(* Logix 5000 project; controller cal1615 1756-L62 rev 20.19; software revision 20.05; part 38 of 82 *)
(* tags used below, declared in another part *)
   AFI : BOOL;   // Always False Bit
   FAULT : BOOL;   // Fault AFI
   HMI : BOOL;   // AFI HMI
   metering_roll_alarm : TIMER;
   metering_roll_close : TIMER;
   p01_param_turret_dia_ft : REAL;
   p01r02_do_green_stack_light_lel : BOOL;   // System Outputs Green Stack Light
   p01r02_do_red_stack_light_LINE : BOOL;
   p01r02_do_yellow_stack_light : BOOL;   // System Outputs Yellow Stack Light
   p01r02_timer_half_second_off : TIMER;   // System Misc Control Timer Second Pulse Off
   p01r02_timer_half_second_on : TIMER;   // System Misc Control Timer 1/2 Second Pulse On
   p01r09_pb_global_reset : BOOL;   // System Modes PB: Global Fault Reset
   p01r13_timer_line_start_warning_dwell : TIMER;   // System Line Start Sequence Pre Start Warning Dwell Timer
   p11r30 : routine;   // Zone 1 Temperature Control
   p12r30 : routine;   // Zone 2 Temperature Control
   p20_acc_ctr_prs_input_max : REAL;
   p20_acc_ctr_prs_input_min : REAL;
   p20_acc_ctr_prs_output_max : REAL;
   p20_acc_ctr_prs_output_min : REAL;
   p20_acc_fill_prs_input_max : REAL;
   p20_acc_fill_prs_input_min : REAL;
   p20_acc_fill_prs_output_max : REAL;
   p20_acc_fill_prs_output_min : REAL;
   p20_acc_ten_prs_input_max : REAL;
   p20_acc_ten_prs_input_min : REAL;
   p20_acc_ten_prs_output_max : REAL;
   p20_acc_ten_prs_output_min : REAL;
   p20_ao_acc_ctr_prs : REAL;   // Letoff Analog Output Accumulator Counter Pressure
   p20_ao_acc_fill_prs : REAL;   // Letoff Analog Output Accumulator Fill Pressure
   p20_ao_acc_ten_prs : REAL;   // Letoff Analog Output Accumulator Tension Pressure
   p20_ao_lo_turret_selected_speed : REAL;   // Letoff Letoff Turret VFD Selected Speed
   p20_ao_loa_selected_speed : REAL;   // Letoff Output Selected Speed
   p20_ao_loa_torque : REAL;
   p20_ao_lob_selected_speed : REAL;   // Letoff Letoff B VFD Selected Speed
   p20_ao_lob_torque : REAL;
   p20_di_acc_empty : BOOL;   // Letoff Digital Input Letoff Accumulator Empty Position
   p20_di_acc_full : BOOL;   // Letoff Digital Input Letoff Accumulator Full Control Position
   p20_di_clutch_prs_ok : BOOL;   // Letoff Modes Accumulator Position Mode
   p20_di_lo_turret : acs800_di_normal;   // Letoff Letoff Turret VFD Drive Inputs
   p20_di_loa_active : BOOL;   // Letoff Digital Input Letoff A Active
   p20_dint_to_hmi : DINT[16];   // Letoff Dint to HMI
   p20_do_acc_enable_tension : BOOL;   // Letoff Digital Output Enable Accumulator Lift Tension
   p20_do_acc_high_prs : BOOL;   // Letoff Digital Output Enable Accumulator Lift Pressure
   p20_do_close_nip : BOOL;   // Letoff Digital Output Feedroll Roll Nip Close
   p20_do_enable_lfr_fwd : BOOL;   // Letoff Digital Output Letoff Accumulator Feedroll Forward
   p20_do_enable_lfr_rev : BOOL;   // Letoff Digital Output Letoff Accumulator Feedroll Reverse
   p20_do_engage_lfr_clutch : BOOL;   // Letoff Digital Output Engage Letoff Accumulator Feedroll Clutch
   p20_do_wdr_turret : acs800_do_normal;
   p20_param_lo_turret_gear_ratio : REAL;
   p20_param_loa_gear_ratio : REAL;
   p20_param_lob_gear_ratio : REAL;
   p20_vfd_di_loa : acs800_di_normal;   // Letoff A VFD Inputs
   p20_vfd_di_lob : acs800_di_normal;   // Letoff B VFD Inputs
   p20_vfd_do_loa : acs800_do_normal;   // Letoff A VFD Outputs
   p20_vfd_do_lob : acs800_do_normal;   // Letoff B VFD Outputs
   p20r01 : routine;   // Letoff Main
   p20r02_letoff_dia_ft : REAL;   // Letoff Misc Control Letoff Diameter [ft]
   p20r04 : routine;   // Letoff Ouput
   p20r04_acc_ctr_prs : SYS_SCP;   // Letoff Analog Outputs Accumulator Counter Pressure
   p20r04_acc_fill_prs : SYS_SCP;   // Letoff Analog Output Accumulator Fill Pressure
   p20r04_acc_ten_prs : SYS_SCP;   // Letoff Analog Output Accumulator Tension Pressure
   p20r04_lo_turret_speed_to_vfd : SYS_SPEED_TO_VFD;   // Letoff Outputs Letoff Turret Speed
   p20r04_loa_speed_to_vfd : SYS_SPEED_TO_VFD;   // Letoff Outputs Letoff A Speed
   p20r04_lob_speed_to_vfd : SYS_SPEED_TO_VFD;   // Letoff Outputs Letoff B Speed
   p20r04_timer_fault : TIMER[4];   // Letoff Output Fault Delay
   p20r04_timer_warning : TIMER[4];   // Letoff Output Warning Delay
   p20r05 : routine;   // Letoff Dint to HMI
   p20r05_timer_fault : TIMER[4];   // Letoff Dint to HMI Fault Delay
   p20r05_timer_warning : TIMER[4];   // Letoff Dint to HMI Warning Delay
   p20r09_accumulator_auto : BOOL;   // Letoff Modes Accumulator Auto Mode
   p20r13_status : DINT;   // Letoff Accumulator Fill Status
   p20r15_loa_on : BOOL;   // Letoff Letoff A VFD On
   p20r16_lob_on : BOOL;   // Letoff Letoff B On
   p20r18_index_complete : BOOL;   // Letoff Letoff Turret VFD Index Complete
   retraction_delay_timer : TIMER;
(* P20_Letoff, continued *)

ROUTINE R04_Output   (* ladder *)
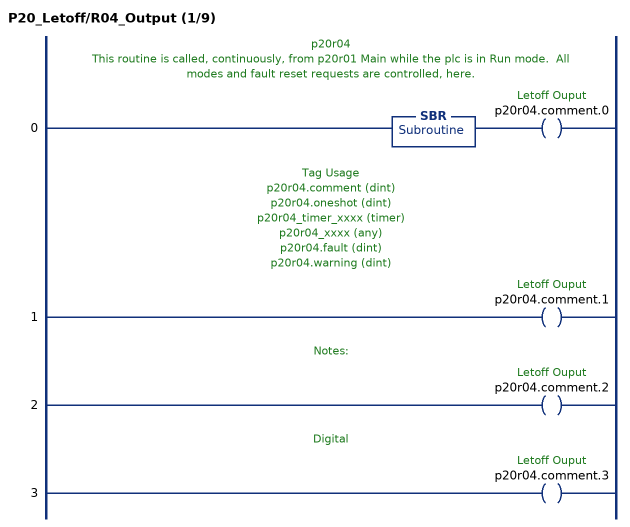
   // p20r04
   // This routine is called, continuously, from p20r01 Main while the plc is in Run mode.  All modes and fault reset requests are controlled, here.
   0: SBR()OTE(p20r04.comment.0);
   // Tag Usage
   // p20r04.comment (dint)
   // p20r04.oneshot (dint)
   // p20r04_timer_xxxx (timer)
   // p20r04_xxxx (any)
   // p20r04.fault (dint)
   // p20r04.warning (dint)
   1: OTE(p20r04.comment.1);
   // Notes:
   2: OTE(p20r04.comment.2);
   // Digital
   3: OTE(p20r04.comment.3);
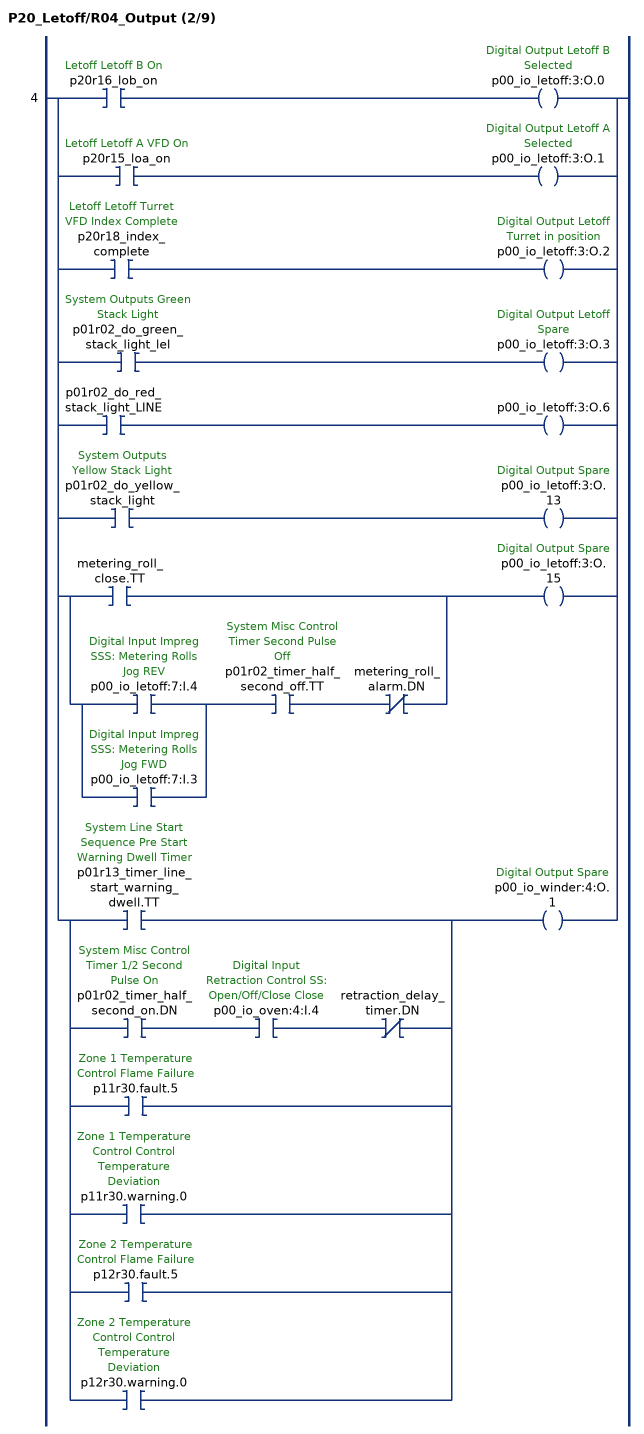
   4: [XIC(p20r16_lob_on) OTE(p00_io_letoff:3:O.0) ,XIC(p20r15_loa_on) OTE(p00_io_letoff:3:O.1) ,XIC(p20r18_index_complete) OTE(p00_io_letoff:3:O.2) ,XIC(p01r02_do_green_stack_light_lel) OTE(p00_io_letoff:3:O.3) ,XIC(p01r02_do_red_stack_light_LINE) OTE(p00_io_letoff:3:O.6) ,[XIC(p01r02_do_yellow_stack_light) OTE(p00_io_letoff:3:O.13) ,[[XIC(metering_roll_close.TT) ,[XIC(p00_io_letoff:7:I.4) ,XIC(p00_io_letoff:7:I.3) ] XIC(p01r02_timer_half_second_off.TT) XIO(metering_roll_alarm.DN) ] OTE(p00_io_letoff:3:O.15) ,[XIC(p01r13_timer_line_start_warning_dwell.TT) ,XIC(p01r02_timer_half_second_on.DN) XIC(p00_io_oven:4:I.4) XIO(retraction_delay_timer.DN) ,XIC(p11r30.fault.5) ,XIC(p11r30.warning.0) ,XIC(p12r30.fault.5) ,XIC(p12r30.warning.0) ] OTE(p00_io_winder:4:O.1) ] ] ];
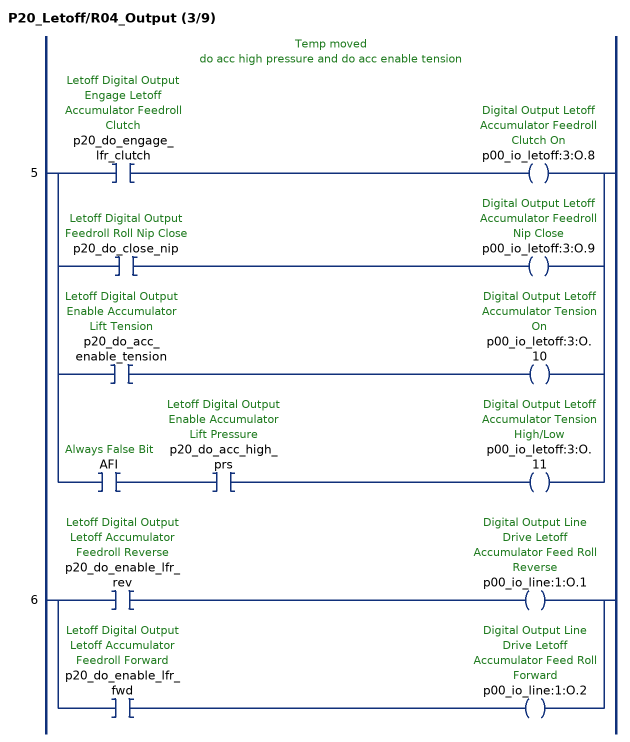
   // Temp moved
   // do acc high pressure and do acc enable tension
   5: [XIC(p20_do_engage_lfr_clutch) OTE(p00_io_letoff:3:O.8) ,XIC(p20_do_close_nip) OTE(p00_io_letoff:3:O.9) ,XIC(p20_do_acc_enable_tension) OTE(p00_io_letoff:3:O.10) ,XIC(AFI) XIC(p20_do_acc_high_prs) OTE(p00_io_letoff:3:O.11) ];
   6: [XIC(p20_do_enable_lfr_rev) OTE(p00_io_line:1:O.1) ,XIC(p20_do_enable_lfr_fwd) OTE(p00_io_line:1:O.2) ];
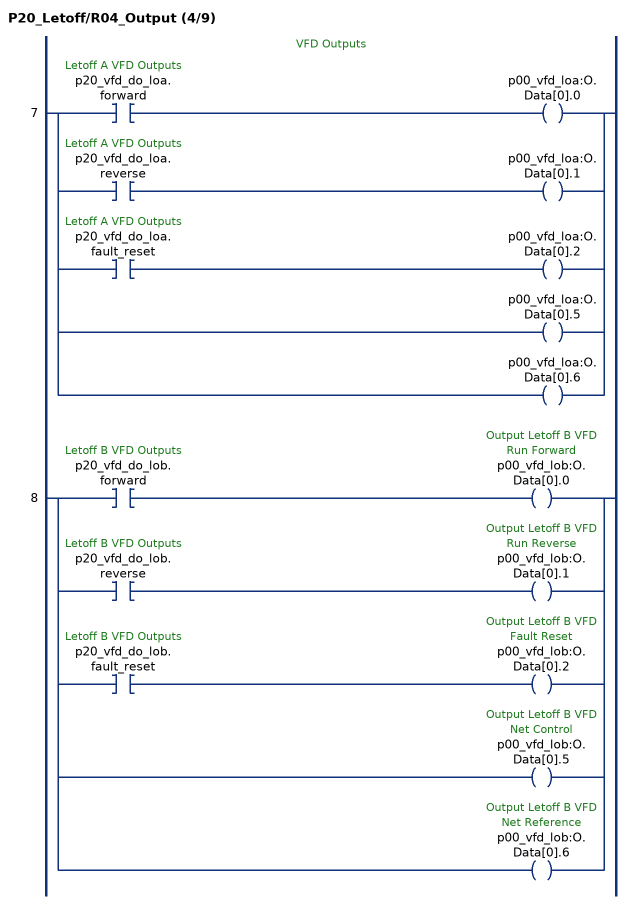
   // VFD Outputs
   7: [XIC(p20_vfd_do_loa.forward) OTE(p00_vfd_loa:O.Data[0].0) ,XIC(p20_vfd_do_loa.reverse) OTE(p00_vfd_loa:O.Data[0].1) ,XIC(p20_vfd_do_loa.fault_reset) OTE(p00_vfd_loa:O.Data[0].2) ,OTE(p00_vfd_loa:O.Data[0].5) ,OTE(p00_vfd_loa:O.Data[0].6) ];
   8: [XIC(p20_vfd_do_lob.forward) OTE(p00_vfd_lob:O.Data[0].0) ,XIC(p20_vfd_do_lob.reverse) OTE(p00_vfd_lob:O.Data[0].1) ,XIC(p20_vfd_do_lob.fault_reset) OTE(p00_vfd_lob:O.Data[0].2) ,OTE(p00_vfd_lob:O.Data[0].5) ,OTE(p00_vfd_lob:O.Data[0].6) ];
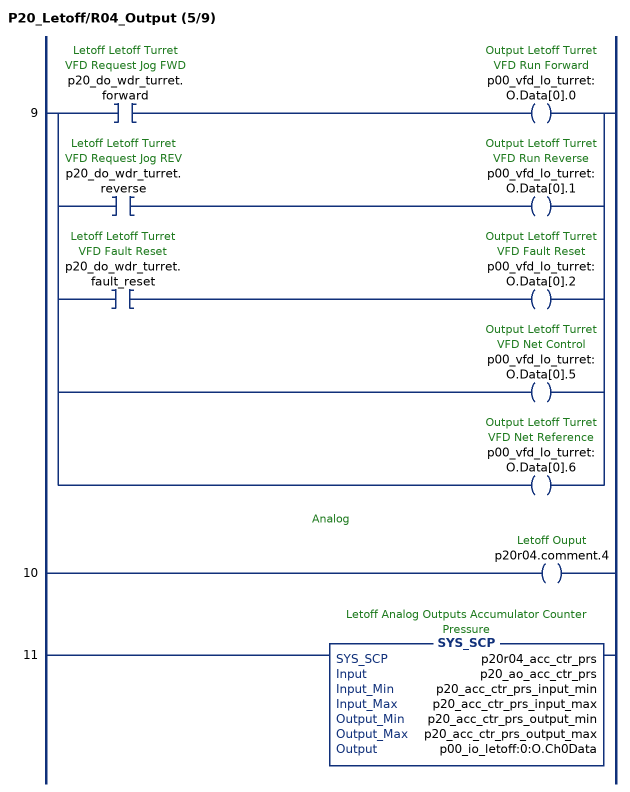
   9: [XIC(p20_do_wdr_turret.forward) OTE(p00_vfd_lo_turret:O.Data[0].0) ,XIC(p20_do_wdr_turret.reverse) OTE(p00_vfd_lo_turret:O.Data[0].1) ,XIC(p20_do_wdr_turret.fault_reset) OTE(p00_vfd_lo_turret:O.Data[0].2) ,OTE(p00_vfd_lo_turret:O.Data[0].5) ,OTE(p00_vfd_lo_turret:O.Data[0].6) ];
   // Analog
   10: OTE(p20r04.comment.4);
   11: SYS_SCP(p20r04_acc_ctr_prs,p20_ao_acc_ctr_prs,p20_acc_ctr_prs_input_min,p20_acc_ctr_prs_input_max,p20_acc_ctr_prs_output_min,p20_acc_ctr_prs_output_max,p00_io_letoff:0:O.Ch0Data);
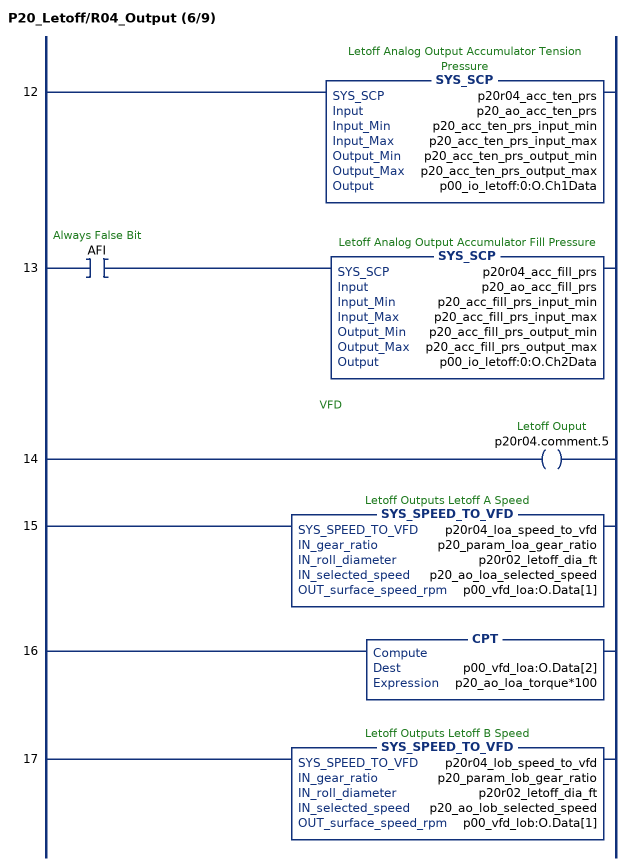
   12: SYS_SCP(p20r04_acc_ten_prs,p20_ao_acc_ten_prs,p20_acc_ten_prs_input_min,p20_acc_ten_prs_input_max,p20_acc_ten_prs_output_min,p20_acc_ten_prs_output_max,p00_io_letoff:0:O.Ch1Data);
   13: XIC(AFI)SYS_SCP(p20r04_acc_fill_prs,p20_ao_acc_fill_prs,p20_acc_fill_prs_input_min,p20_acc_fill_prs_input_max,p20_acc_fill_prs_output_min,p20_acc_fill_prs_output_max,p00_io_letoff:0:O.Ch2Data);
   // VFD
   14: OTE(p20r04.comment.5);
   15: SYS_SPEED_TO_VFD(p20r04_loa_speed_to_vfd,p20_param_loa_gear_ratio,p20r02_letoff_dia_ft,p20_ao_loa_selected_speed,p00_vfd_loa:O.Data[1]);
   16: CPT(p00_vfd_loa:O.Data[2],p20_ao_loa_torque*100);
   17: SYS_SPEED_TO_VFD(p20r04_lob_speed_to_vfd,p20_param_lob_gear_ratio,p20r02_letoff_dia_ft,p20_ao_lob_selected_speed,p00_vfd_lob:O.Data[1]);
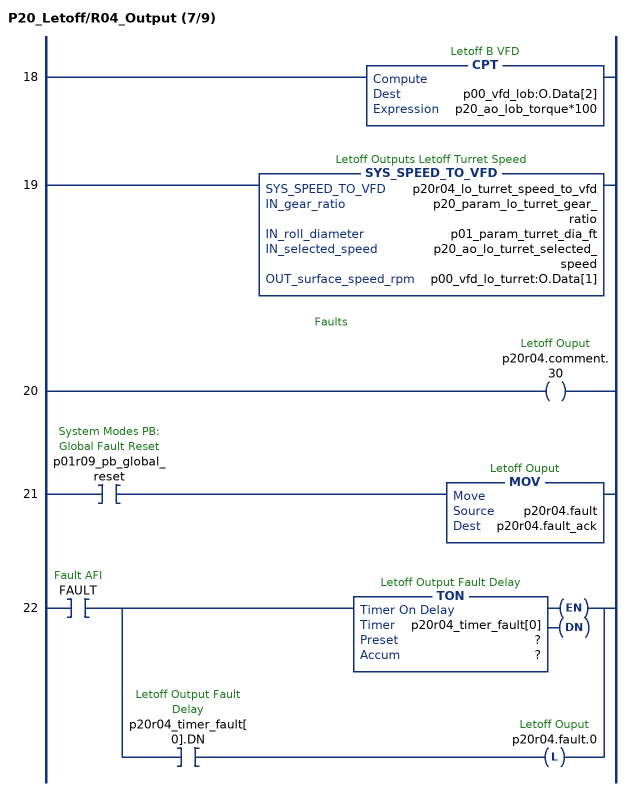
   18: CPT(p00_vfd_lob:O.Data[2],p20_ao_lob_torque*100);
   19: SYS_SPEED_TO_VFD(p20r04_lo_turret_speed_to_vfd,p20_param_lo_turret_gear_ratio,p01_param_turret_dia_ft,p20_ao_lo_turret_selected_speed,p00_vfd_lo_turret:O.Data[1]);
   // Faults
   20: OTE(p20r04.comment.30);
   21: XIC(p01r09_pb_global_reset)MOV(p20r04.fault,p20r04.fault_ack);
   22: XIC(FAULT)[TON(p20r04_timer_fault[0],?,?) ,XIC(p20r04_timer_fault[0].DN) OTL(p20r04.fault.0) ];
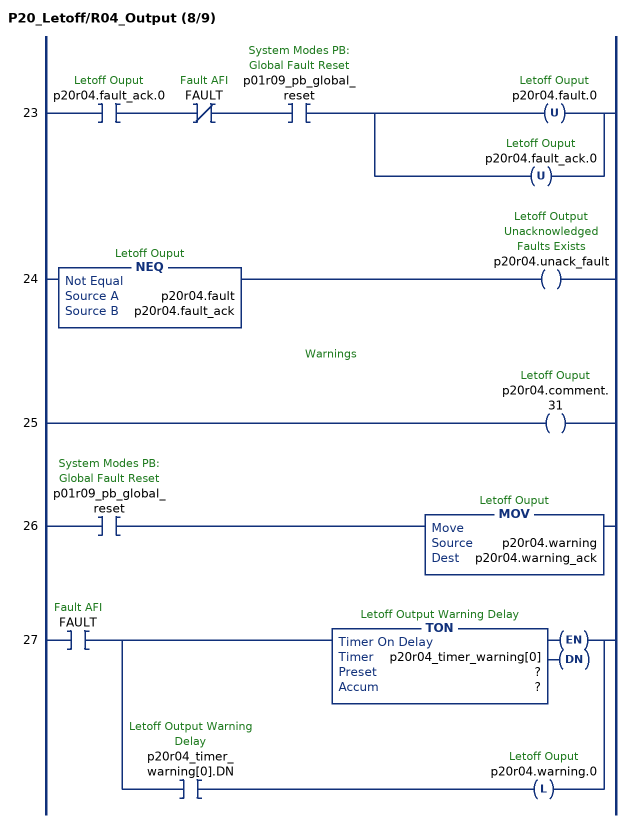
   23: XIC(p20r04.fault_ack.0)XIO(FAULT)XIC(p01r09_pb_global_reset)[OTU(p20r04.fault.0) ,OTU(p20r04.fault_ack.0) ];
   24: NEQ(p20r04.fault,p20r04.fault_ack)OTE(p20r04.unack_fault);
   // Warnings
   25: OTE(p20r04.comment.31);
   26: XIC(p01r09_pb_global_reset)MOV(p20r04.warning,p20r04.warning_ack);
   27: XIC(FAULT)[TON(p20r04_timer_warning[0],?,?) ,XIC(p20r04_timer_warning[0].DN) OTL(p20r04.warning.0) ];
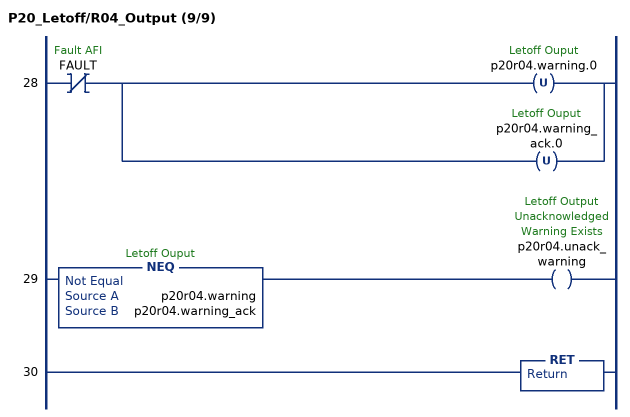
   28: XIO(FAULT)[OTU(p20r04.warning.0) ,OTU(p20r04.warning_ack.0) ];
   29: NEQ(p20r04.warning,p20r04.warning_ack)OTE(p20r04.unack_warning);
   30: RET();
END_ROUTINE

ROUTINE R05_Dint_to_HMI   (* ladder *)
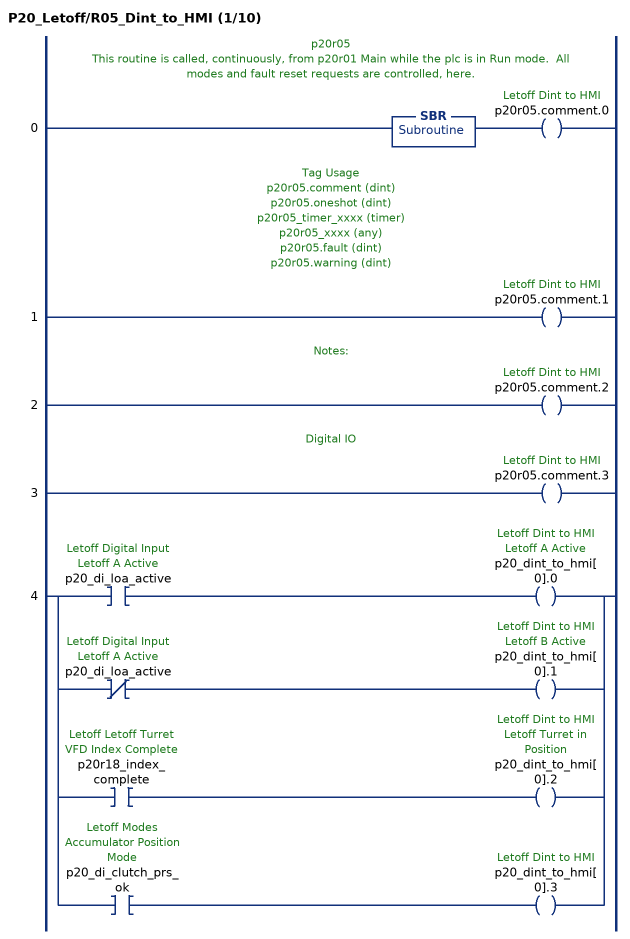
   // p20r05
   // This routine is called, continuously, from p20r01 Main while the plc is in Run mode.  All modes and fault reset requests are controlled, here.
   0: SBR()OTE(p20r05.comment.0);
   // Tag Usage
   // p20r05.comment (dint)
   // p20r05.oneshot (dint)
   // p20r05_timer_xxxx (timer)
   // p20r05_xxxx (any)
   // p20r05.fault (dint)
   // p20r05.warning (dint)
   1: OTE(p20r05.comment.1);
   // Notes:
   2: OTE(p20r05.comment.2);
   // Digital IO
   3: OTE(p20r05.comment.3);
   4: [XIC(p20_di_loa_active) OTE(p20_dint_to_hmi[0].0) ,XIO(p20_di_loa_active) OTE(p20_dint_to_hmi[0].1) ,XIC(p20r18_index_complete) OTE(p20_dint_to_hmi[0].2) ,XIC(p20_di_clutch_prs_ok) OTE(p20_dint_to_hmi[0].3) ];
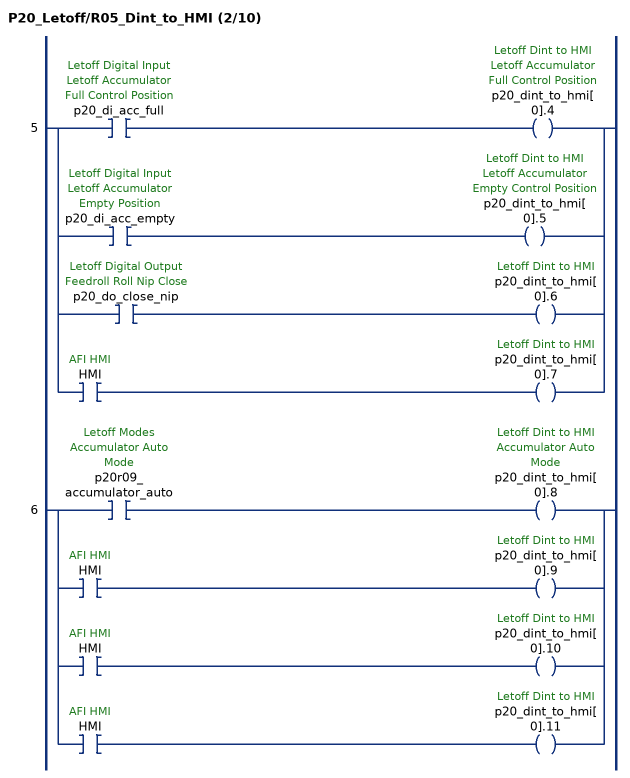
   5: [XIC(p20_di_acc_full) OTE(p20_dint_to_hmi[0].4) ,XIC(p20_di_acc_empty) OTE(p20_dint_to_hmi[0].5) ,XIC(p20_do_close_nip) OTE(p20_dint_to_hmi[0].6) ,XIC(HMI) OTE(p20_dint_to_hmi[0].7) ];
   6: [XIC(p20r09_accumulator_auto) OTE(p20_dint_to_hmi[0].8) ,XIC(HMI) OTE(p20_dint_to_hmi[0].9) ,XIC(HMI) OTE(p20_dint_to_hmi[0].10) ,XIC(HMI) OTE(p20_dint_to_hmi[0].11) ];
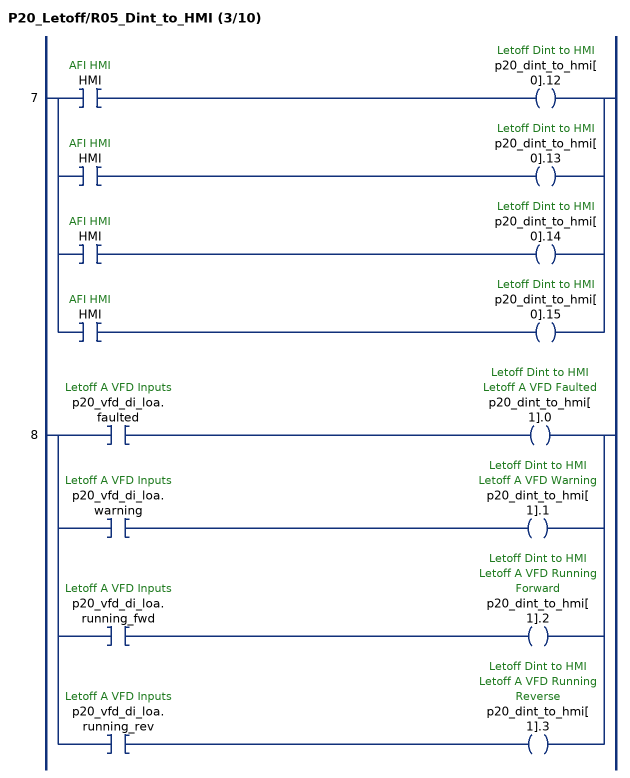
   7: [XIC(HMI) OTE(p20_dint_to_hmi[0].12) ,XIC(HMI) OTE(p20_dint_to_hmi[0].13) ,XIC(HMI) OTE(p20_dint_to_hmi[0].14) ,XIC(HMI) OTE(p20_dint_to_hmi[0].15) ];
   8: [XIC(p20_vfd_di_loa.faulted) OTE(p20_dint_to_hmi[1].0) ,XIC(p20_vfd_di_loa.warning) OTE(p20_dint_to_hmi[1].1) ,XIC(p20_vfd_di_loa.running_fwd) OTE(p20_dint_to_hmi[1].2) ,XIC(p20_vfd_di_loa.running_rev) OTE(p20_dint_to_hmi[1].3) ];
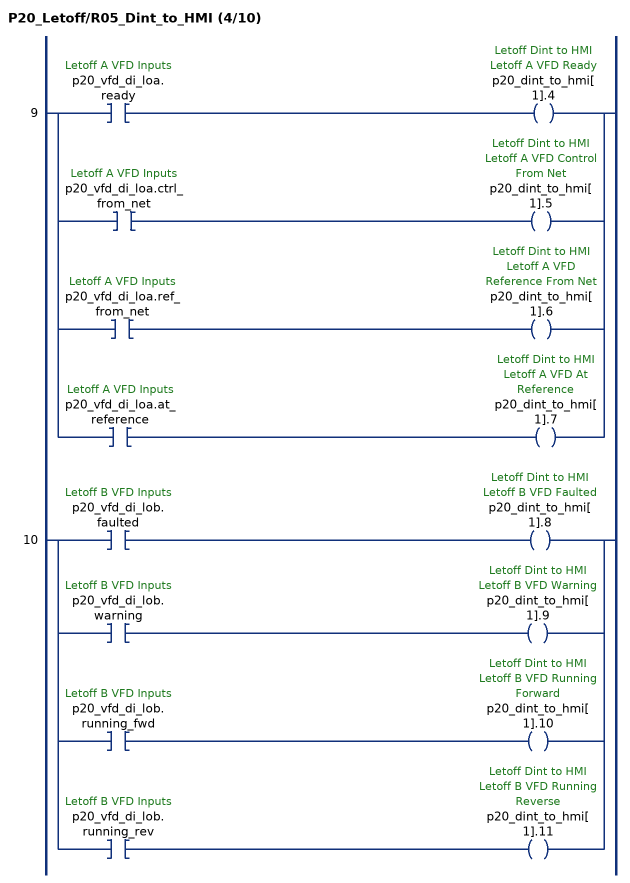
   9: [XIC(p20_vfd_di_loa.ready) OTE(p20_dint_to_hmi[1].4) ,XIC(p20_vfd_di_loa.ctrl_from_net) OTE(p20_dint_to_hmi[1].5) ,XIC(p20_vfd_di_loa.ref_from_net) OTE(p20_dint_to_hmi[1].6) ,XIC(p20_vfd_di_loa.at_reference) OTE(p20_dint_to_hmi[1].7) ];
   10: [XIC(p20_vfd_di_lob.faulted) OTE(p20_dint_to_hmi[1].8) ,XIC(p20_vfd_di_lob.warning) OTE(p20_dint_to_hmi[1].9) ,XIC(p20_vfd_di_lob.running_fwd) OTE(p20_dint_to_hmi[1].10) ,XIC(p20_vfd_di_lob.running_rev) OTE(p20_dint_to_hmi[1].11) ];
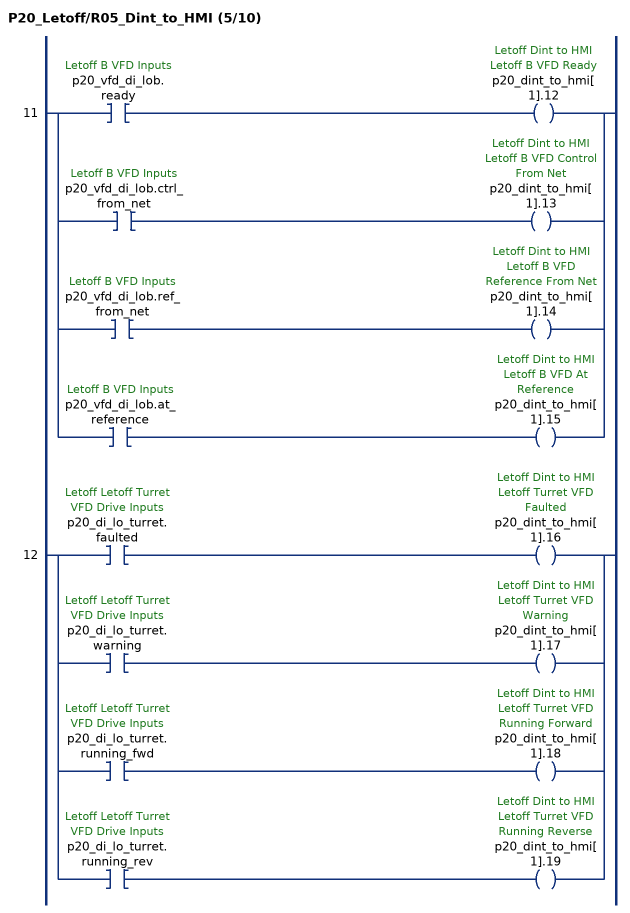
   11: [XIC(p20_vfd_di_lob.ready) OTE(p20_dint_to_hmi[1].12) ,XIC(p20_vfd_di_lob.ctrl_from_net) OTE(p20_dint_to_hmi[1].13) ,XIC(p20_vfd_di_lob.ref_from_net) OTE(p20_dint_to_hmi[1].14) ,XIC(p20_vfd_di_lob.at_reference) OTE(p20_dint_to_hmi[1].15) ];
   12: [XIC(p20_di_lo_turret.faulted) OTE(p20_dint_to_hmi[1].16) ,XIC(p20_di_lo_turret.warning) OTE(p20_dint_to_hmi[1].17) ,XIC(p20_di_lo_turret.running_fwd) OTE(p20_dint_to_hmi[1].18) ,XIC(p20_di_lo_turret.running_rev) OTE(p20_dint_to_hmi[1].19) ];
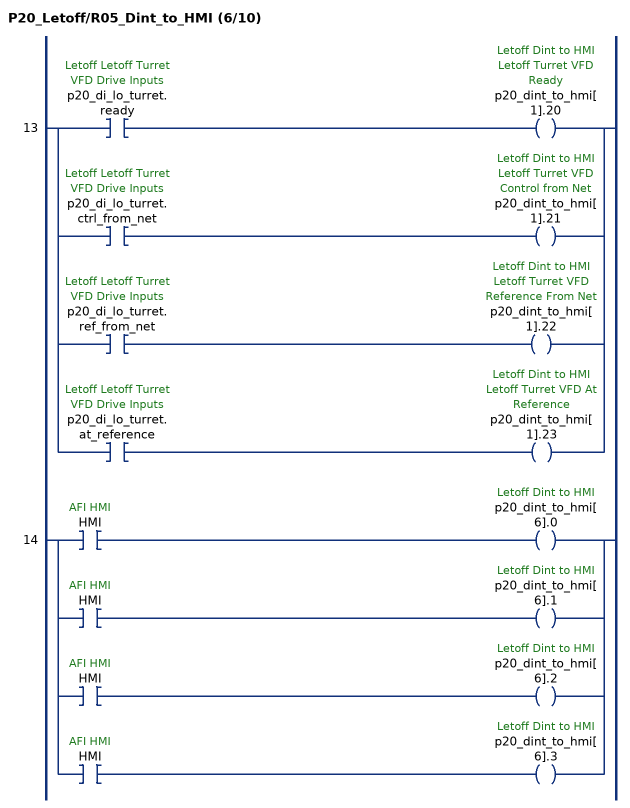
   13: [XIC(p20_di_lo_turret.ready) OTE(p20_dint_to_hmi[1].20) ,XIC(p20_di_lo_turret.ctrl_from_net) OTE(p20_dint_to_hmi[1].21) ,XIC(p20_di_lo_turret.ref_from_net) OTE(p20_dint_to_hmi[1].22) ,XIC(p20_di_lo_turret.at_reference) OTE(p20_dint_to_hmi[1].23) ];
   14: [XIC(HMI) OTE(p20_dint_to_hmi[6].0) ,XIC(HMI) OTE(p20_dint_to_hmi[6].1) ,XIC(HMI) OTE(p20_dint_to_hmi[6].2) ,XIC(HMI) OTE(p20_dint_to_hmi[6].3) ];
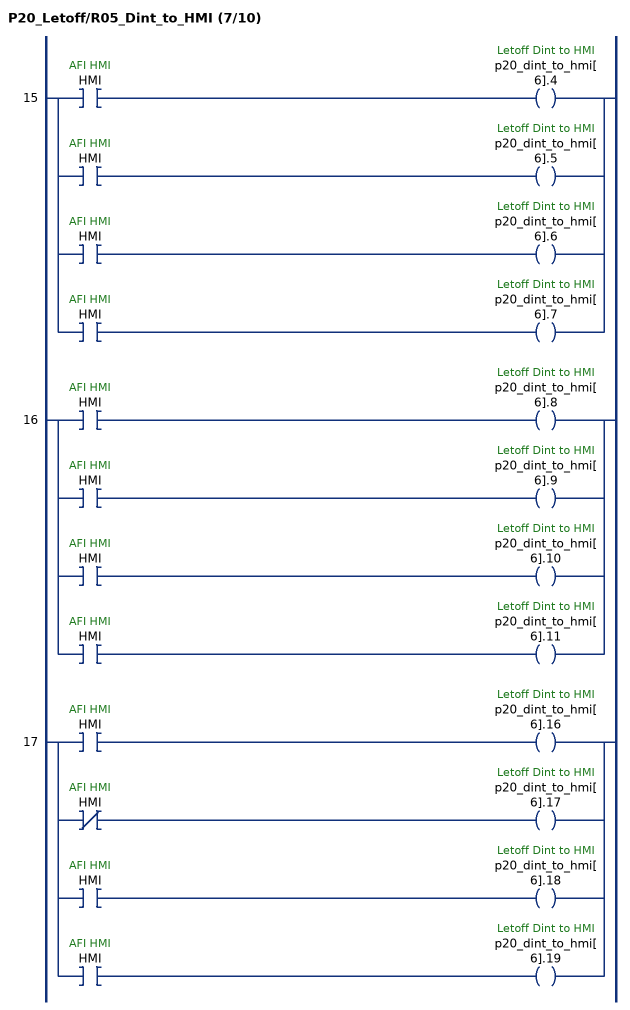
   15: [XIC(HMI) OTE(p20_dint_to_hmi[6].4) ,XIC(HMI) OTE(p20_dint_to_hmi[6].5) ,XIC(HMI) OTE(p20_dint_to_hmi[6].6) ,XIC(HMI) OTE(p20_dint_to_hmi[6].7) ];
   16: [XIC(HMI) OTE(p20_dint_to_hmi[6].8) ,XIC(HMI) OTE(p20_dint_to_hmi[6].9) ,XIC(HMI) OTE(p20_dint_to_hmi[6].10) ,XIC(HMI) OTE(p20_dint_to_hmi[6].11) ];
   17: [XIC(HMI) OTE(p20_dint_to_hmi[6].16) ,XIO(HMI) OTE(p20_dint_to_hmi[6].17) ,XIC(HMI) OTE(p20_dint_to_hmi[6].18) ,XIC(HMI) OTE(p20_dint_to_hmi[6].19) ];
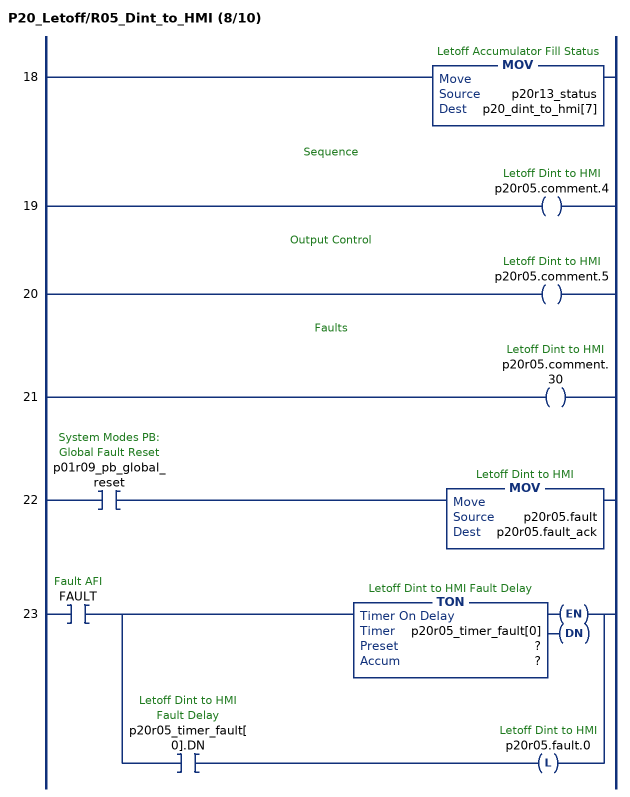
   18: MOV(p20r13_status,p20_dint_to_hmi[7]);
   // Sequence
   19: OTE(p20r05.comment.4);
   // Output Control
   20: OTE(p20r05.comment.5);
   // Faults
   21: OTE(p20r05.comment.30);
   22: XIC(p01r09_pb_global_reset)MOV(p20r05.fault,p20r05.fault_ack);
   23: XIC(FAULT)[TON(p20r05_timer_fault[0],?,?) ,XIC(p20r05_timer_fault[0].DN) OTL(p20r05.fault.0) ];
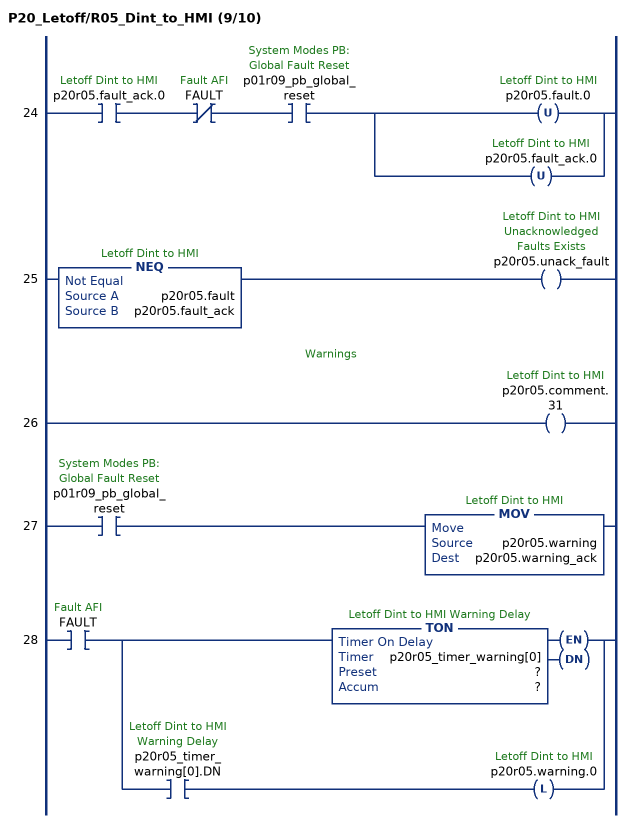
   24: XIC(p20r05.fault_ack.0)XIO(FAULT)XIC(p01r09_pb_global_reset)[OTU(p20r05.fault.0) ,OTU(p20r05.fault_ack.0) ];
   25: NEQ(p20r05.fault,p20r05.fault_ack)OTE(p20r05.unack_fault);
   // Warnings
   26: OTE(p20r05.comment.31);
   27: XIC(p01r09_pb_global_reset)MOV(p20r05.warning,p20r05.warning_ack);
   28: XIC(FAULT)[TON(p20r05_timer_warning[0],?,?) ,XIC(p20r05_timer_warning[0].DN) OTL(p20r05.warning.0) ];
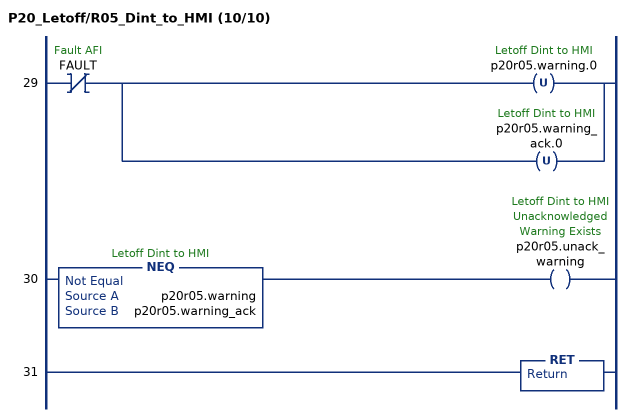
   29: XIO(FAULT)[OTU(p20r05.warning.0) ,OTU(p20r05.warning_ack.0) ];
   30: NEQ(p20r05.warning,p20r05.warning_ack)OTE(p20r05.unack_warning);
   31: RET();
END_ROUTINE
